(*
SPDX-FileCopyrightText: © 2026 Oleksandr Tiutyk <trofimich@gmail.com>
SPDX-License-Identifier: MIT
License: https://opensource.org/license/mit
*)

(*!
<summary>
Describes an automation component that exposes children, dispatches broadcasts and provides action
permissions.
</summary>
<description>
Permission requests are evaluated locally and then through parents; the first rejection ends evaluation.
Each child in the execution hierarchy occupies one slot and identifies its containing branch as Parent.
Other components may borrow the same child independently of this hierarchy.
Indexed Try lookups return borrowed interfaces or null and do not propagate exceptions.
</description>
*)
INTERFACE IParentAutomationComponent EXTENDS IAutomationComponent, TOF_Core.IActionPermissionProvider

{attribute 'monitoring' := 'call'}
PROPERTY FINAL ActionPermissionPolicy : TOF_Core.IActionPermissionPolicy
GET
END_GET
SET
END_SET
END_PROPERTY

{attribute 'monitoring' := 'call'}
PROPERTY ChildCount : TOF_Core.INT_LENGTH
GET
END_GET
END_PROPERTY

{attribute 'monitoring' := 'call'}
PROPERTY FINAL ChildCriticalErrorHandlingPolicy : IChildCriticalErrorHandlingPolicy
GET
END_GET
SET
END_SET
END_PROPERTY

METHOD GetEffectiveChildCriticalErrorHandlingPolicy : IChildCriticalErrorHandlingPolicy
END_METHOD

(*!
<summary>Requests permission from this level and its parents, stopping at the first rejection.</summary>
<description>
A missing policy permits its level; the request succeeds only if no level rejects it. The
IActionPermissionProvider contract applies: live non-null inputs, synchronous borrowing, current rejectReason
on FALSE, ignored rejectReason on TRUE, and propagation of evaluation exceptions.
</description>
*)

METHOD RequestActionPermission : BOOL
VAR_INPUT
	actionDescriptor : TOF_Core.INamed;
	requestingObject : TOF_Core.IObject;
END_VAR
VAR_IN_OUT
	rejectReason : WSTRING(255);
END_VAR
END_METHOD

(*!
<summary>Returns a borrowed child by its zero-based index.</summary>
<description>
Returns null when the entry is unavailable, the index is out of range or a nested call raises an exception.
Fatal allocation observations return null and leave the fatal latch set for the outer task boundary.
Does not transfer ownership or extend lifetime. Implementations must not propagate exceptions.
</description>
*)
METHOD TryGetChildByIndex : IChildAutomationComponent
VAR_INPUT
	index : TOF_Core.INT_INDEX;
END_VAR
END_METHOD

END_INTERFACE

(* stored: Version 1.1.0.1
   Itf IParentAutomationComponent: Id {07b4e225-a246-4050-a6a8-78b85fbf51d5}
   Property ActionPermissionPolicy: Id {670eab9e-aaa6-4bf4-887e-46068ed7503b}
   Get Get: Id {968f8af4-7f9e-4cde-9a57-9d309dd69c73}
   Set Set: Id {f69466ed-f037-47de-9949-934c657aef01}
   Property ChildCount: Id {00ca3c22-be54-413b-ae6c-1b5517138933}
   Get Get: Id {459b2cc0-c67e-4878-a038-92f034e9cc37}
   Property ChildCriticalErrorHandlingPolicy: Id {a0b08b12-4afb-4708-b8da-01cbec5556c3}
   Get Get: Id {0ff7e562-90a8-4ef0-be5a-88bbf12688b1}
   Set Set: Id {f5cf81a1-da1b-4aee-a7d5-7973b76dd488}
   Method GetEffectiveChildCriticalErrorHandlingPolicy: Id {5af06bb0-07ff-4210-9e37-c7cd3950ec29}
   Method RequestActionPermission: Id {357b341e-acea-4699-b246-83e901e17844}
   Method TryGetChildByIndex: Id {da4ea733-d5b7-445d-932a-6ee0bac437e7} *)
